TYPE ST_HMICommand :
STRUCT
    eCommandType : E_CommandType;
    nAxisIndex : UINT;
    fValue1 : LREAL;
    fValue2 : LREAL;
    eTargetMode : E_MachineMode;
    nAlarmID : UINT;
    bExecute : BOOL;
END_STRUCT
END_TYPE

(* stored: Version 1.1.0.1
   DUT ST_HMICommand: Id {B174C1F5-6B87-7924-596A-75A8832BB142} *)
